{attribute 'GeneratedUsingTerminal: EQ3314-0002-0016'}
{attribute addProperty BoxType "EQ3314-0002-0016"}
{attribute addProperty Id "TC_TCInputs_Channel_1AT %I*TC_TCInputs_Channel_A8DF64E310TC_TCInputs_Channel_2AT %I*TC_TCInputs_Channel_A8DF64E310TC_TCInputs_Channel_3AT %I*TC_TCInputs_Channel_A8DF64E310TC_TCInputs_Channel_4AT %I*TC_TCInputs_Channel_A8DF64E310WcStateAT %I*WcState_9091E0EB2InfoDataAT %I*InfoData_94A18F5E2"}
{attribute addProperty CRC "251088390"}
{attribute addProperty Size "44"}
TYPE EQ3314_0EF74E06 EXTENDS EtcSlaveTerminalBase_947E5A46 :
STRUCT
	{attribute addProperty Name "TC_TCInputs_Channel_1"}
	TC_TCInputs_Channel_1 : TC_TCInputs_Channel_A8DF64E3;
	{attribute addProperty Name "TC_TCInputs_Channel_2"}
	TC_TCInputs_Channel_2 : TC_TCInputs_Channel_A8DF64E3;
	{attribute addProperty Name "TC_TCInputs_Channel_3"}
	TC_TCInputs_Channel_3 : TC_TCInputs_Channel_A8DF64E3;
	{attribute addProperty Name "TC_TCInputs_Channel_4"}
	TC_TCInputs_Channel_4 : TC_TCInputs_Channel_A8DF64E3;
	{attribute addProperty Name "WcState"}
	WcState : WcState_9091E0EB;
	{attribute addProperty Name "InfoData"}
	InfoData : InfoData_94A18F5E;
END_STRUCT
END_TYPE

(* stored: Version 1.2.0.0, ProductVersion 3.1.4024.9
   DUT EQ3314_0EF74E06: Id {25d0a08d-3593-4f01-ad83-f5fda6ff4857} *)
